RoboDK station: Duplo_Builder.rdk

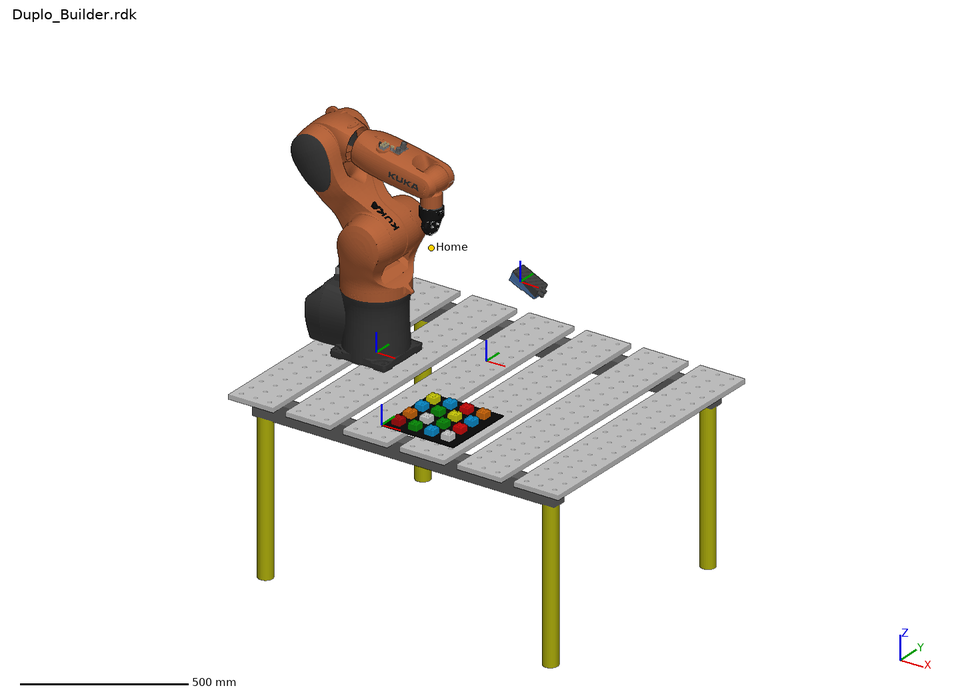
[picture v0: the station drawn from its stored meshes, robots at their saved joint values, targets as dots, program paths as lines]
Station Duplo_Builder (saved by RoboDK 5.2.1). Poses are relative to the parent item; angles as X-Y-Z fixed-axis rotations.
Station parameters (name, value as stored): IO_5, 1
  - frame World at (0, 0, 0) mm
    - object Table at (400, 0, 0) mm, size 1193.8 x 965.2 x 609.6 mm, geometry from welding_table.sld
    - target Home (Cartesian target) at (200, 0, 400) mm; joints [0, -127.181, 137.503, 0, 79.677, -90] of KUKA KR 6 R700 sixx
  - frame KUKA KR 6 R700 sixx Base at (0, 0, 0) mm
    - robot KUKA KR 6 R700 sixx: 6 axes, payload 6 kg, reach 706.7 mm, repeatability 0.03 mm, weight 50 kg
        modified DH rows (alpha deg, a mm, theta deg, d mm): 0, 0, 0, 400; -90, 25, 0, 0; 0, 315, -90, 0; -90, 35, 0, 365; 90, 0, 0, 0; -90, 0, 180, 80
        joint limits [-170, -190, -120, -185, -120, -350] to [170, 45, 156, 185, 120, 350]; home [0, -90, 90, 0, 0, 0]; saved at [0, -127.181, 137.503, 0, 79.677, -90]
      - robot RobotiQ 2F85: 1 axes, payload 5 kg
          joint limits [0] to [85]; home [85]; saved at [0]
      - tool GripperTCP, TCP at (0, 0, 140) mm, rotated rx -180 ry 0 rz 90 deg
  - frame LegoBricks at (300, -400, 5) mm
    - object Plate at (260, 0, -5) mm, size 260 x 260 x 5 mm, geometry from Plate.step
    - object Brick 4 at (20, 80, 0) mm, size 32 x 32 x 24 mm, geometry from Brick.step
    - object Brick 3 at (200, 80, 0) mm, size 32 x 32 x 24 mm, geometry from Brick.step
    - object Brick 3 at (140, 200, 0) mm, size 32 x 32 x 24 mm, geometry from Brick.step
    - object Brick 3 at (80, 200, 0) mm, size 32 x 32 x 24 mm, geometry from Brick.step
    - object Brick 3 at (20, 200, 0) mm, size 32 x 32 x 24 mm, geometry from Brick.step
    - object Brick 7 at (20, 140, 0) mm, size 32 x 32 x 24 mm, geometry from Brick.step
    - object Brick 3 at (200, 200, 0) mm, size 32 x 32 x 24 mm, geometry from Brick.step
    - object Brick 5 at (80, 80, 0) mm, size 32 x 32 x 24 mm, geometry from Brick.step
    - object Brick 3 at (200, 20, 0) mm, size 32 x 32 x 24 mm, geometry from Brick.step
    - object Brick 1 at (20, 20, 0) mm, size 32 x 32 x 24 mm, geometry from Brick.step
    - object Brick 2 at (80, 20, 0) mm, size 32 x 32 x 24 mm, geometry from Brick.step
    - object Brick 6 at (140, 80, 0) mm, size 32 x 32 x 24 mm, geometry from Brick.step
    - object Brick 8 at (80, 140, 0) mm, size 32 x 32 x 24 mm, geometry from Brick.step
    - object Brick 9 at (140, 140, 0) mm, size 32 x 32 x 24 mm, geometry from Brick.step
    - object Brick 3 at (200, 140, 0) mm, size 32 x 32 x 24 mm, geometry from Brick.step
    - object Brick 3 at (140, 20, 0) mm, size 32 x 32 x 24 mm, geometry from Brick.step
  - frame LEGOBuilder at (300, 140, 0) mm
  - frame CameraCoord at (710, -270, 540) mm
    - object Camera at (0, 0, 0) mm, rotated rx 180 ry -25 rz 180 deg, size 53 x 116 x 38 mm, geometry from Cam2D_SICK_VSPP_5F2113.sld
  - program Reset (1 instructions, listed below)

--- program Reset (robot KUKA KR 6 R700 sixx) ---
  Replace objects
